(* PLC project Unnamed, Unknown Unnamed 1 *)
(* stored: creationDateTime 2023-10-24T08:11:18, modificationDateTime 2023-12-04T14:28:20 *)

PROGRAM UAS_PLC
  VAR
    START : BOOL;
    STOP : BOOL;
    CR_MOTOR1 : BOOL;
    MOTOR_PUMP1 : BOOL;
    LEVEL_SWITCH2 : BOOL;
    LEVEL_SWITCH1 : BOOL;
    CR_LEVEL1 : BOOL;
    CR_LEVEL2 : BOOL;
    PL1 : BOOL;
    PL2 : BOOL;
    CR1 : BOOL;
    CR2 : BOOL;
    SOLENOID_VALVE1 : BOOL;
    SOLENOID_VALVE2 : BOOL;
  END_VAR

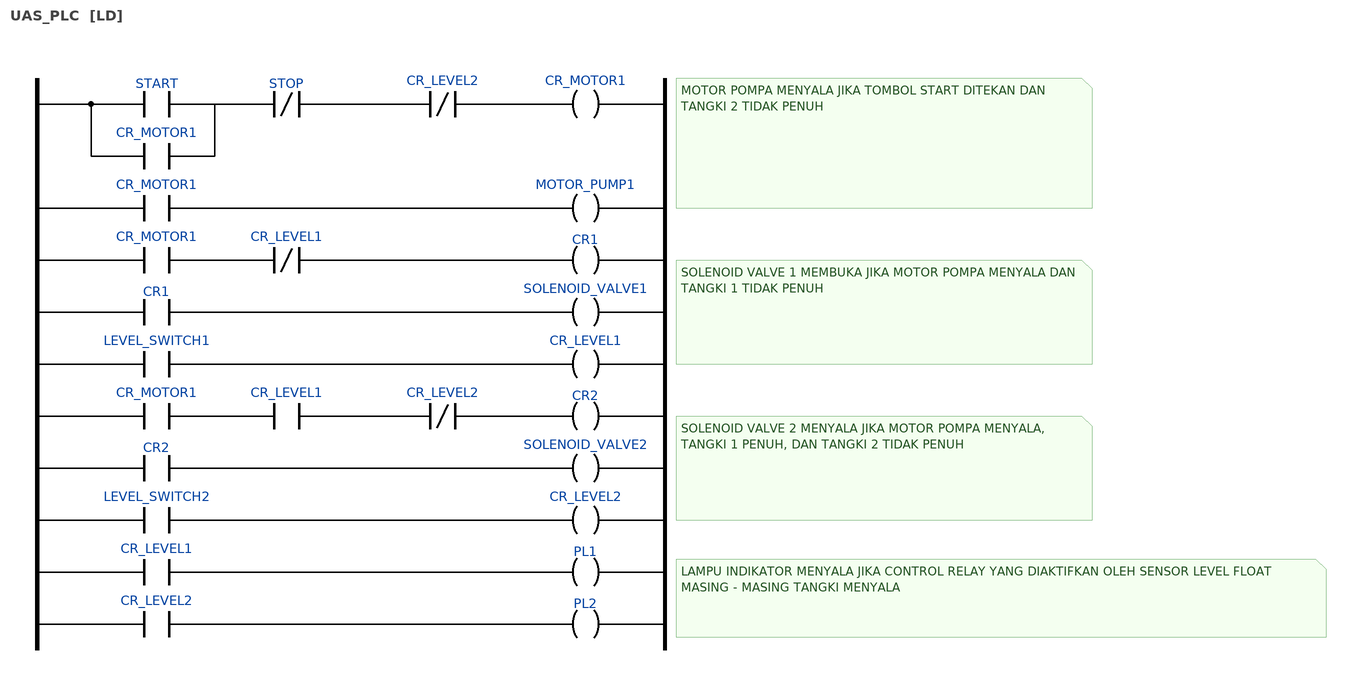
(* LD diagram, written out as Structured Text *)
(* MOTOR POMPA MENYALA JIKA TOMBOL START DITEKAN DAN TANGKI 2 TIDAK PENUH *)
CR_MOTOR1 := (START OR CR_MOTOR1) AND NOT STOP AND NOT CR_LEVEL2;
MOTOR_PUMP1 := CR_MOTOR1;
CR1 := CR_MOTOR1 AND NOT CR_LEVEL1;
(* SOLENOID VALVE 1 MEMBUKA JIKA MOTOR POMPA MENYALA DAN TANGKI 1 TIDAK PENUH *)
SOLENOID_VALVE1 := CR1;
CR_LEVEL1 := LEVEL_SWITCH1;
CR2 := CR_MOTOR1 AND CR_LEVEL1 AND NOT CR_LEVEL2;
(* SOLENOID VALVE 2 MENYALA JIKA MOTOR POMPA MENYALA, TANGKI 1 PENUH, DAN TANGKI 2 TIDAK PENUH *)
SOLENOID_VALVE2 := CR2;
CR_LEVEL2 := LEVEL_SWITCH2;
(* LAMPU INDIKATOR MENYALA JIKA CONTROL RELAY YANG DIAKTIFKAN OLEH SENSOR LEVEL FLOAT MASING - MASING TANGKI MENYALA *)
PL1 := CR_LEVEL1;
PL2 := CR_LEVEL2;
END_PROGRAM

CONFIGURATION Config0
  RESOURCE Res0 ON PLC
    TASK task0(INTERVAL := T#20ms, PRIORITY := 0);
    PROGRAM instance0 WITH task0 : UAS_PLC;
  END_RESOURCE
END_CONFIGURATION
